TEXTLIST AxesMoveProcessUnitsTextList
  0 = 'd / m / s'
  1 = 'degrees'
  2 = 'arcmin'
  3 = 'arcsec'
  4 = 'rad'
   = ''
END_TEXTLIST

(* stored: Version 1.1.0.1, ProductVersion 3.1.4019.2
   TextList AxesMoveProcessUnitsTextList: Id {7921ab72-9332-497b-add0-5878539d34b2} *)
